// Monitors the dump chiller from the flow sensor
FUNCTION_BLOCK FB_DumpChiller
VAR_INPUT
	bAmphosOn : BOOL; // Whether the amphos is turned on
	bDumpChillerFlow : BOOL; // Signal from the flow sensor. Normally high.
END_VAR
VAR_OUTPUT
	{attribute 'pytmc' := '
		pv: ERROR
		io: i
		field: OSV MAJOR
		field: ZSV NO_ALARM
		field: ZNAM OK
		field: ONAM ERROR
	'}
	bError : BOOL; // Whether an error was detected. Latches until reset
END_VAR
VAR
END_VAR

(* Latch error if the dump chiller flow detects an error and the amphos is on *)
IF bAmphosOn AND NOT bDumpChillerFlow THEN
	bError := TRUE;
END_IF

// Reset latched errors
METHOD Reset
VAR_INPUT
END_VAR
bError := FALSE;
END_METHOD

END_FUNCTION_BLOCK

(* stored: Version 1.1.0.1, ProductVersion 3.1.4020.14
   POU FB_DumpChiller: Id {116e5a5e-5390-4f77-a571-6eef4757f21f}, SpecialFunc None
   Method Reset: Id {798c5e10-f7ad-4fe8-969f-0ab4a0d7941b} *)
